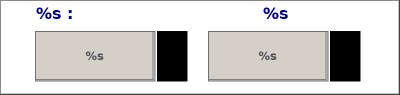
VISUALIZATION SA_VERIN  // 400x95
VAR_IN_OUT
	m_Input_VERIN : BLOCK_ACTUATOR;
END_VAR
    RoundedRectangle (0,0 400x95), text variable: m_Input_VERIN.MNEMO
    RoundedRectangle (157,31 30x50), colour toggle: m_Input_VERIN.STATE_ON
    Button (35,31 120x50), "%s", input disabled if: NOT m_Input_VERIN.Autor_On_IHM OR NOT m_Input_VERIN.MANUAL OR NOT (PRG_User.ACTU_USER.FONCTION_SA AND NOT MACHINE.STATE_PROD), text list: 'TextList_Orders', text index: 3
        tap m_Input_VERIN.M_ON
    RoundedRectangle (330,31 30x50), colour toggle: m_Input_VERIN.STATE_Off
    Button (208,31 120x50), "%s", input disabled if: NOT m_Input_VERIN.Autor_Off_IHM OR NOT m_Input_VERIN.MANUAL OR NOT (PRG_User.ACTU_USER.FONCTION_SA AND NOT MACHINE.STATE_PROD), text list: 'TextList_Orders', text index: 2
        tap m_Input_VERIN.M_OFF
    Rectangle (33,3 247x21), "%s :", text list: 'TextList_Actuator_Type', text index: 0
    Rectangle (260,3 119x21), "%s", text variable: m_Input_VERIN.MNEMO
END_VISUALIZATION

(* stored: Version 1.1.0.1, ProductVersion 3.1.4024.10
   Visu SA_VERIN: Id {3cbdc0a8-d8da-4722-bce9-e9a9372624ae} *)
